KUKA KRL program: caldejgen.src

&ACCESS RV1
&REL 190
&COMMENT Funcion de calculo de dejadas
DEF CalDejGen()

  ;*************************************************;
  ;***    CALCULAR POSICION DE DEJADA EN PALE    ***;
  ;                                                 ;
  ; Creacion de los mosaicos para las producciones. ;
  ;                                                 ;
  ; Salidas:                                        ;
  ;   XAPROX - Posicion de aproximacion a la dejada.;
  ;   XDEJ   - Posicion de dejada.                  ;
  ;   XSAL   - Posicion de salida de la dejada.     ;
  ;*************************************************;

  ; TipoProducto = 1

  ; TipoPalet = 1  ->  Europal
  ; TipoPalet = 2  ->  Especifico

  ; Dato = 1  ->  NumeroCajas
  ; Dato = 2  ->  TipoCogida
  ; Dato = 3  ->  CintaCogida 1

  ; TipoCogida = 1  ->  Pala fija vallado
  ; TipoCogida = 2  ->  No se contempla

  ; CintaCogida = 1  ->  Entrada

  ; Giro = 1 -> Abre hacia CONTRARIO Robot
  ; Giro = 2 -> Abre hacia CONTRARIO entrada producto

  ; CapayPosicionActual  ->  Ajuste de capa y posicion actual
  ; Posicion+Paridad  ->  Capa impar 1-10
  ; Posicion+Paridad  ->  Capa par 11-20


  MaximoCapas=DatosProduccion[Produccion_Actual,1]
  MAXIMAPOSICION = DatosProduccion[Produccion_Actual,2]
  TIPOPRODUCTO=DatosProduccion[Produccion_Actual,3]
  TIPOPALE=DatosProduccion[Produccion_Actual,4]
  ANCHOPRODUCTO =DatosSaco[TIPOPRODUCTO,1]
  LARGOPRODUCTO = DatosSaco[TIPOPRODUCTO,2]
  ALTOPRODUCTO = DatosSaco[TIPOPRODUCTO,3]
  ANCHOPALE =DatosPale[TipoPale,1]
  LARGOPALE = DatosPale[TipoPale,2]
  ALTOPALE = DatosPale[TipoPale,3]


  POSICIONX = DATOSDEJADA[Produccion_Actual, CAPAYPOSICION_ACTUAL_1, 1]
  POSICIONY = DATOSDEJADA[Produccion_Actual, CAPAYPOSICION_ACTUAL_1, 2]
  GIRO = DATOSDEJADA[Produccion_Actual, CAPAYPOSICION_ACTUAL_1, 3]
  TIPO_COGIDA = DATOSDEJADA[Produccion_Actual, CAPAYPOSICION_ACTUAL_1, 4]

  AJUSTEX = 0
  AJUSTEY = 0
  AJUSTEZ = 165

    ORIGENPALEX = 0
    ORIGENPALEY = 0
    ORIGENPALEZ = 0




    IF NOT LIMITE_CAPAS_DARSENA1 THEN
        DARSENA1=TRUE
        DARSENA2=FALSE
    ELSE
        DARSENA1=FALSE
        DARSENA2=TRUE
    ENDIF





    XDEJADA.X = POSICIONX + ORIGENPALEX + AJUSTEX
    XDEJADA.Y = POSICIONY + ORIGENPALEY + AJUSTEY


IF DARSENA1 THEN
      XDEJADA.Z = (CONTADOR_CAPAS_DARSENA1)*ALTOPRODUCTO + ORIGENPALEZ + AJUSTEZ
ENDIF

IF DARSENA2 THEN
      XDEJADA.Z = (CONTADOR_CAPAS_DARSENA2)*ALTOPRODUCTO + ORIGENPALEZ + AJUSTEZ
ENDIF


    XDEJADA.A = -180
    XDEJADA.B = 0


;EN PRODUCCION CONJUNTA DAMOS PRIORIDAD A LA DARSENA 1
;CUANDO SE LLENE, PASAMOS A LA DARSENA 2
;SI NO ES PRODUCCION CONJUNTA-->DARSENA 1





;ORIENTACION DE DEJADA
;DEPENDIENDO DE LA DARSENA, ESTE ANGULO CAMBIARÁ Y EL TIPO DE CODIDA TAMBI�?N

SWITCH GIRO

  CASE 1



          IF DARSENA1 THEN

              XDEJADA.A=-90
              XDEJADA.C=-180

              XDEJADA.T=58
              XDEJADA.S=6

          ELSE

            SWITCH TIPO_COGIDA

              CASE 1
                  TIPO_COGIDA=3
              CASE 2
                  TIPO_COGIDA=4
              CASE 3
                  TIPO_COGIDA=1
              CASE 4
                  TIPO_COGIDA=2
              ENDSWITCH


              XDEJADA.A=90
              XDEJADA.C = 0

              XDEJADA.T=58
              XDEJADA.S=6

          ENDIF


  CASE 2

            IF DARSENA1 THEN

                  XDEJADA.A=0
                  XDEJADA.C = -180

                  XDEJADA.T=58
                  XDEJADA.S=6


            ELSE

              SWITCH TIPO_COGIDA

                          CASE 1
                              TIPO_COGIDA=3
                          CASE 2
                              TIPO_COGIDA=4
                          CASE 3
                              TIPO_COGIDA=1
                          CASE 4
                              TIPO_COGIDA=2
                          ENDSWITCH


                          XDEJADA.A=180
                          XDEJADA.C = 0

                          XDEJADA.T=58
                          XDEJADA.S=6
            ENDIF

  CASE 3


    IF DARSENA1 THEN

                    XDEJADA.A=90
                    XDEJADA.C = -180

                    XDEJADA.T=26
                    XDEJADA.S=6

   ELSE

                    SWITCH TIPO_COGIDA

                                      CASE 1
                                          TIPO_COGIDA=3
                                      CASE 2
                                          TIPO_COGIDA=4
                                      CASE 3
                                          TIPO_COGIDA=1
                                      CASE 4
                                          TIPO_COGIDA=2
                    ENDSWITCH





                                  XDEJADA.A=-90
                                  XDEJADA.C = 0

                                  XDEJADA.T=58
                                  XDEJADA.S=6

ENDIF

ENDSWITCH


    XAPROXIMACION_DEJADA = XDEJADA

    XAPROXIMACION_DEJADA.X= XDEJADA.X - 100
    XAPROXIMACION_DEJADA.Y= XDEJADA.Y - 100
    XAPROXIMACION_DEJADA.Z= XDEJADA.Z + 250


    ;PUNTO SALIDA - MISMO PUNTO MÁS EL ALTO DEL SACO
    XSALIDA_DEJADA = XDEJADA
    XSALIDA_DEJADA.Z = XDEJADA.Z + ALTOproducto +30





end
